PROGRAM MAIN
VAR
END_VAR

(* 
	GOF 		Define the skeleton of an algorithm in an operation, deferring some steps to subclasses.
				Template method lets subclasses redefine certain steps of an algorithm without changing 
				the algorithm's structure. 
*)
P_TemplateMethod();

END_PROGRAM

(* stored: Version 1.1.0.1, ProductVersion 3.1.4024.12
   POU MAIN: Id {f66ea7df-ba2b-41b6-890c-d7c0d96d098c}, SpecialFunc None *)
